// TIA Portal V16 export
// export: Created 2024-12-03T15:41:40.9894445Z, ExportSetting WithDefaults, DisplayName Totally Integrated Automation Portal, DisplayVersion V16 Update 6, DisplayName TIA Portal Version Control Interface, DisplayVersion V16 Update 2, DisplayName TIA Portal Openness, DisplayVersion V16 Update 6, DisplayName TIA Portal Teamcenter Gateway, DisplayVersion V16, DisplayName SINAMICS Startdrive Advanced, DisplayVersion V16 Update 5, DisplayName SINAMICS Startdrive G130, G150, S120, S150, SINAMICS MV, S210, DisplayVersion V16 Update 5, DisplayName SINAMICS Startdrive G110M, G120, G120C, G120D, G120P, G115D, DisplayVersion V16 Update 5, DisplayName STEP 7 Professional, DisplayVersion V16 Update 6, DisplayName STEP 7 Safety, DisplayVersion V16, DisplayName WinCC Advanced / Unified PC, DisplayVersion V16 Update 6
FUNCTION_BLOCK "SmartBool"   // FB21, SCL
{ S7_Optimized_Access := 'FALSE' }
VERSION : 0.1
// stored: AutoNumber true, IsIECCheckEnabled false, SetENOAutomatically false, UDAEnableTagReadback false
   VAR_INPUT
      I_Sensor : Bool;
      I_Simulate : Bool;
      HoldOnTIme : Time;
      DelayOnTime : Time;
   END_VAR
   VAR_OUTPUT
      O_data : "SmartBooldt";
   END_VAR
   VAR DB_SPECIFIC
      S_Prev_Val : Bool;
      S_DelayOnTime { S7_SetPoint := 'True'} : TON_TIME;
      S_HoldOnTimer { ExternalAccessible := 'False'; ExternalVisible := 'False'; ExternalWritable := 'False'; S7_SetPoint := 'True'} : TOF_TIME;
      S_LE : Bool;
      S_FE : Bool;
      S_SensorState : Bool;
      S_HoldOn : Bool;
   END_VAR
   VAR_TEMP
      T_Signal : Bool;
   END_VAR
BEGIN


   IF #DelayOnTime = t#0ms THEN
       #T_Signal := #I_Sensor OR #I_Simulate;
   ELSE

       #S_DelayOnTime(IN:=#I_Sensor OR #I_Simulate,
                      PT:=#DelayOnTime,
                      Q=>#T_Signal);

   END_IF;

   #S_HoldOnTimer(IN := #T_Signal,
                PT := #HoldOnTIme,
                Q => #S_HoldOn);

   #S_SensorState := #S_HoldOn;

   //Leading edge
   IF #S_SensorState AND NOT #S_Prev_Val THEN
       #S_LE := true;

   ELSE
       #S_LE := FALSE;

   END_IF;

   //Falling edge
   IF NOT #S_SensorState AND #S_Prev_Val THEN
       #S_FE := true;
   ELSE
       #S_FE := false;
   END_IF;


   #S_Prev_Val := #S_HoldOn;

   //Transfer output
   #O_data.State := #S_SensorState ;
   #O_data.FE := #S_FE;
   #O_data.LE := #S_LE;

   //Counter
   //
   IF #O_data.LE THEN
       #O_data.Counter += 1;
   END_IF;

   IF "HMI_DB".ResetSensorCounters.signal THEN
       #O_data.Counter := 0;
   END_IF;
END_FUNCTION_BLOCK
